TYPE U_OdriveIntBytes :
UNION
    Value : INT;
    Bytes : ARRAY[0..1] OF BYTE;
END_UNION
END_TYPE

(* stored: Version 1.1.0.1
   DUT U_OdriveIntBytes: Id {1CC68910-4ED4-490C-9F0B-A80EB5630F48} *)
